// TIA Portal project "Projet_charg_bout" (V15)

(* hardware
DEVICE "PC-System_1"  SIMATIC PC station
   slot 0: "Station PC SIMATIC"  Rail  SIMATIC PC-Station  V1.0
      slot 125: "Stationmanager"  Station_Manager  V6.0.4
   slot 1: "HMI_RT_1"  WinCC RT Advanced  6AV2 104-0xxxx-xxxx  15.0.0.0
      slot 33792: "Interface hôte"  Host interface
   slot 2: "IE Général_1"  IE General  IE_CP  V8.2.0
DEVICE "Station S7-1200_1"  S7-1200 Station
   slot 0: "Châssis_0"  S7-1200 Rack  Rack  V1.0
   slot 1: "PLC_1"  CPU 1214C AC/DC/Rly  6ES7 214-1BG40-0XB0  V4.2
*)

// ===== PLC "PLC_1"  CPU 1214C AC/DC/Rly =====

VAR_GLOBAL   // PLC tag table "Table de variables standard"
   "Tag_1" AT %M100.0 : Bool;
END_VAR

VAR_GLOBAL   // PLC tag table "INPUT"
   "I_GHT" AT %I0.0 : Bool;
   "I_GHD" AT %I0.1 : Bool;
   "I_CB_CHAT" AT %I0.2 : Bool;
   "BI_START" AT %I0.3 : Bool;
   "I_CB_CHAT_TRONG_KET" AT %I0.4 : Bool;
   "M_GHT" AT %M0.0 : Bool;
   "M_GHD" AT %M0.1 : Bool;
   "M_CB_CHAT" AT %M0.2 : Bool;
   "BM_START" AT %M0.3 : Bool;
   "M_CB_CHAT_TRONG_KET" AT %M0.4 : Bool;
   "BM_SIMULATION" AT %M0.5 : Bool;
   "BM_RESET" AT %M0.6 : Bool;
END_VAR

VAR_GLOBAL   // PLC tag table "OUTPUT"
   "Q_VAN_XA" AT %Q0.0 : Bool;
   "Q_HA" AT %Q0.1 : Bool;
   "Q_NAGA" AT %Q0.2 : Bool;
   "Q_BT" AT %Q0.3 : Bool;
   "Q_FULL" AT %Q0.4 : Bool;
END_VAR

VAR_GLOBAL   // PLC tag table "MANU_NHO"
   "DEM_CHAI" AT %MW100 : Int;
   "SIMU_CHAI_CO" AT %MW102 : Int;
   "SIMU_CTAY" AT %MW104 : Int;
   "DEM_CHI_ROT" AT %MW106 : Int;
   "SIMU_CHAI_DA_ROT" AT %MW108 : Int;
END_VAR

VAR_GLOBAL   // PLC tag table "DELAY_TIME"
   "BIT_DELAT_1S" AT %M10.0 : Bool;
   "BIT_DELAY_1S_1" AT %M10.1 : Bool;
   "BIT_DELAY_1S_2" AT %M10.2 : Bool;
   "BIT_DELAY_1S_3" AT %M10.3 : Bool;
   "SIMU_CHAI_SP_CD" AT %M10.4 : Bool;
END_VAR

VAR_GLOBAL   // PLC tag table "LENH_pandn"
   "P1" AT %M20.0 : Bool;
   "P2" AT %M20.1 : Bool;
   "BIT=1" AT %M20.2 : Bool;
   "P3" AT %M20.3 : Bool;
   "P4" AT %M20.4 : Bool;
   "P5" AT %M20.5 : Bool;
   "P6" AT %M20.6 : Bool;
   "P7" AT %M20.7 : Bool;
   "P8" AT %M21.0 : Bool;
   "P9" AT %M21.1 : Bool;
   "P10" AT %M21.2 : Bool;
   "P11" AT %M21.3 : Bool;
   "P12" AT %M21.4 : Bool;
   "N1" AT %M21.5 : Bool;
   "N2" AT %M21.6 : Bool;
   "P13" AT %M21.7 : Bool;
   "P14" AT %M22.0 : Bool;
END_VAR

// folder: System blocks/Program resources

DATA_BLOCK "IEC_Timer_0_DB"   // DB1
{ S7_Optimized_Access := 'TRUE' }
AUTHOR : Simatic
FAMILY : IEC
NAME : IEC_TMR
VERSION : 1.0
// stored: InstanceOfName IEC_TIMER
"IEC_TIMER"
BEGIN
END_DATA_BLOCK

DATA_BLOCK "IEC_Timer_0_DB_1"   // DB2
{ S7_Optimized_Access := 'TRUE' }
AUTHOR : Simatic
FAMILY : IEC
NAME : IEC_TMR
VERSION : 1.0
// stored: InstanceOfName IEC_TIMER
"IEC_TIMER"
BEGIN
END_DATA_BLOCK

DATA_BLOCK "IEC_Timer_0_DB_2"   // DB3
{ S7_Optimized_Access := 'TRUE' }
AUTHOR : Simatic
FAMILY : IEC
NAME : IEC_TMR
VERSION : 1.0
// stored: InstanceOfName IEC_TIMER
"IEC_TIMER"
BEGIN
END_DATA_BLOCK

DATA_BLOCK "IEC_Timer_0_DB_3"   // DB4
{ S7_Optimized_Access := 'TRUE' }
AUTHOR : Simatic
FAMILY : IEC
NAME : IEC_TMR
VERSION : 1.0
// stored: InstanceOfName IEC_TIMER
"IEC_TIMER"
BEGIN
END_DATA_BLOCK

DATA_BLOCK "IEC_Timer_0_DB_4"   // DB5
{ S7_Optimized_Access := 'TRUE' }
AUTHOR : Simatic
FAMILY : IEC
NAME : IEC_TMR
VERSION : 1.0
// stored: InstanceOfName IEC_TIMER
"IEC_TIMER"
BEGIN
END_DATA_BLOCK

DATA_BLOCK "IEC_Timer_0_DB_5"   // DB6
{ S7_Optimized_Access := 'TRUE' }
AUTHOR : Simatic
FAMILY : IEC
NAME : IEC_TMR
VERSION : 1.0
// stored: InstanceOfName IEC_TIMER
"IEC_TIMER"
BEGIN
END_DATA_BLOCK

DATA_BLOCK "IEC_Timer_0_DB_6"   // DB7
{ S7_Optimized_Access := 'TRUE' }
AUTHOR : Simatic
FAMILY : IEC
NAME : IEC_TMR
VERSION : 1.0
// stored: InstanceOfName IEC_TIMER
"IEC_TIMER"
BEGIN
END_DATA_BLOCK

// folder: (top level)

FUNCTION "FC_SUMILATION" : Void   // FC1, LAD
{ S7_Optimized_Access := 'TRUE' }
VERSION : 0.1
   VAR_TEMP   // added for the SCL form of the ladder/FBD networks
      _w1 : Bool;
   END_VAR
BEGIN

REGION Network 1
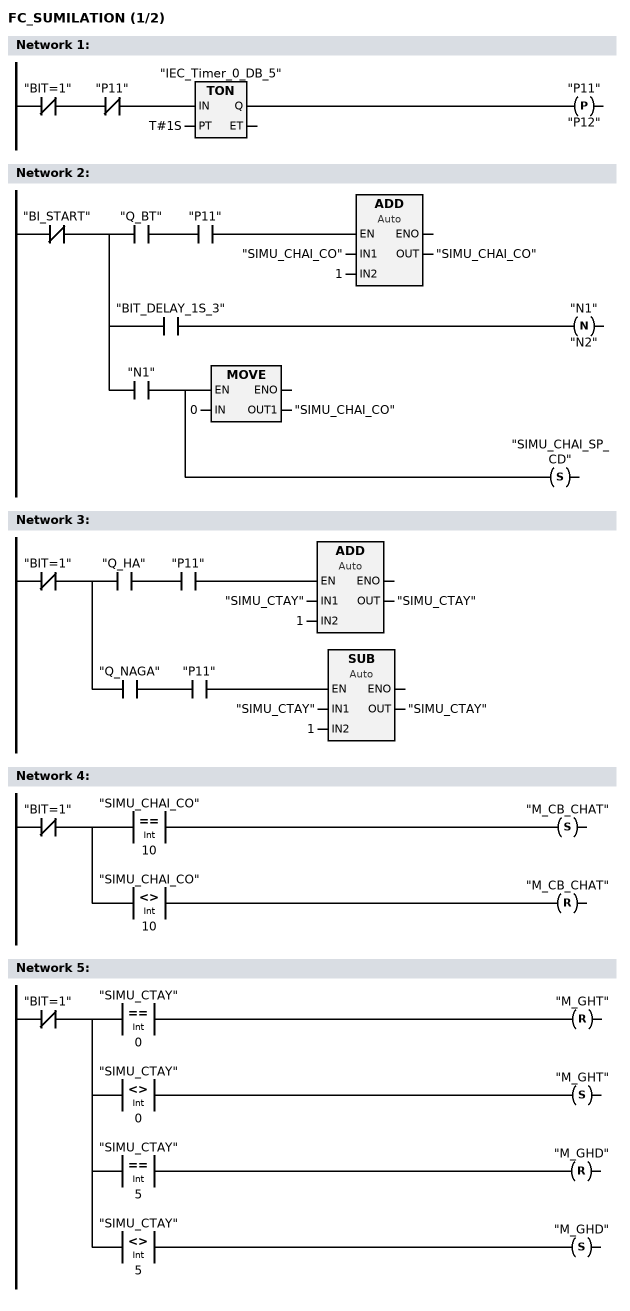
   "IEC_Timer_0_DB_5".TON(IN := NOT "BIT=1" AND NOT "P11", PT := T#1S);
   "P11" := "IEC_Timer_0_DB_5".Q AND NOT "P12";   // rising edge
   "P12" := "IEC_Timer_0_DB_5".Q;
END_REGION

REGION Network 2
   IF NOT "BI_START" AND "Q_BT" AND "P11" THEN "SIMU_CHAI_CO" := "SIMU_CHAI_CO" + 1; END_IF;
   #_w1 := NOT "BI_START" AND "BIT_DELAY_1S_3";
   "N1" := NOT #_w1 AND "N2";   // falling edge
   "N2" := #_w1;
   IF NOT "BI_START" AND "N1" THEN
       "SIMU_CHAI_CO" := 0;
       "SIMU_CHAI_SP_CD" := TRUE;
   END_IF;
END_REGION

REGION Network 3
   RUNG wire#powerrail
      I_Contact( "BIT=1" )
      wire#w1
      Contact( "Q_HA" )
      Contact( "P11" )
      Add(in1 := "SIMU_CTAY", in2 := 1, out => "SIMU_CTAY")
   END_RUNG
   RUNG wire#w1
      Contact( "Q_NAGA" )
      Contact( "P11" )
      Sub(in1 := "SIMU_CTAY", in2 := 1, out => "SIMU_CTAY")
   END_RUNG
   // the same network as SCL:
   IF NOT "BIT=1" AND "Q_HA" AND "P11" THEN "SIMU_CTAY" := "SIMU_CTAY" + 1; END_IF;
   IF NOT "BIT=1" AND "Q_NAGA" AND "P11" THEN "SIMU_CTAY" := "SIMU_CTAY" - 1; END_IF;
END_REGION

REGION Network 4
   RUNG wire#powerrail
      I_Contact( "BIT=1" )
      wire#w1
      { S7_Templates := "SrcType := Int" } EQ_Contact(in1 := "SIMU_CHAI_CO", in2 := 10)
      S_Coil( "M_CB_CHAT" )
   END_RUNG
   RUNG wire#w1
      { S7_Templates := "SrcType := Int" } NE_Contact(in1 := "SIMU_CHAI_CO", in2 := 10)
      R_Coil( "M_CB_CHAT" )
   END_RUNG
   // the same network as SCL:
   IF NOT "BIT=1" AND ("SIMU_CHAI_CO" = 10) THEN "M_CB_CHAT" := TRUE; END_IF;
   IF NOT "BIT=1" AND ("SIMU_CHAI_CO" <> 10) THEN "M_CB_CHAT" := FALSE; END_IF;
END_REGION

REGION Network 5
   RUNG wire#powerrail
      I_Contact( "BIT=1" )
      wire#w1
      { S7_Templates := "SrcType := Int" } EQ_Contact(in1 := "SIMU_CTAY", in2 := 0)
      R_Coil( "M_GHT" )
   END_RUNG
   RUNG wire#w1
      { S7_Templates := "SrcType := Int" } NE_Contact(in1 := "SIMU_CTAY", in2 := 0)
      S_Coil( "M_GHT" )
   END_RUNG
   RUNG wire#w1
      { S7_Templates := "SrcType := Int" } EQ_Contact(in1 := "SIMU_CTAY", in2 := 5)
      R_Coil( "M_GHD" )
   END_RUNG
   RUNG wire#w1
      { S7_Templates := "SrcType := Int" } NE_Contact(in1 := "SIMU_CTAY", in2 := 5)
      S_Coil( "M_GHD" )
   END_RUNG
   // the same network as SCL:
   IF NOT "BIT=1" AND ("SIMU_CTAY" = 0) THEN "M_GHT" := FALSE; END_IF;
   IF NOT "BIT=1" AND ("SIMU_CTAY" <> 0) THEN "M_GHT" := TRUE; END_IF;
   IF NOT "BIT=1" AND ("SIMU_CTAY" = 5) THEN "M_GHD" := FALSE; END_IF;
   IF NOT "BIT=1" AND ("SIMU_CTAY" <> 5) THEN "M_GHD" := TRUE; END_IF;
END_REGION

REGION Network 6
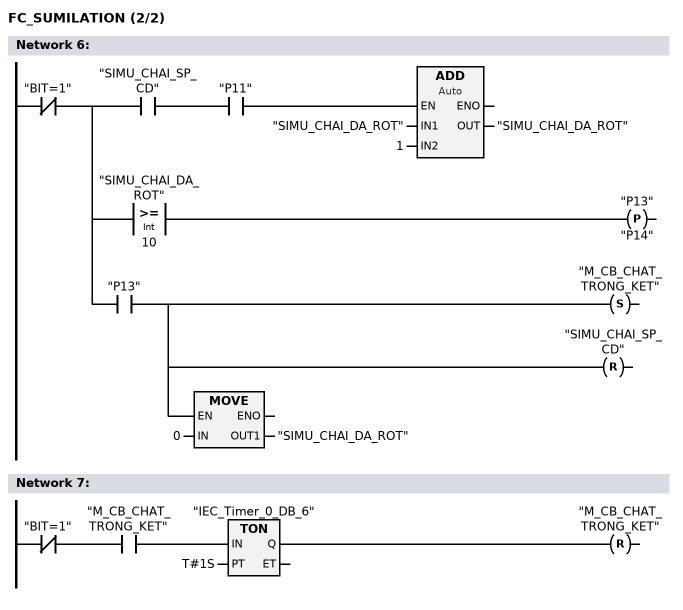
   IF NOT "BIT=1" AND "SIMU_CHAI_SP_CD" AND "P11" THEN "SIMU_CHAI_DA_ROT" := "SIMU_CHAI_DA_ROT" + 1; END_IF;
   #_w1 := NOT "BIT=1" AND ("SIMU_CHAI_DA_ROT" >= 10);
   "P13" := #_w1 AND NOT "P14";   // rising edge
   "P14" := #_w1;
   IF NOT "BIT=1" AND "P13" THEN
       "M_CB_CHAT_TRONG_KET" := TRUE;
       "SIMU_CHAI_SP_CD" := FALSE;
       "SIMU_CHAI_DA_ROT" := 0;
   END_IF;
END_REGION

REGION Network 7
   "IEC_Timer_0_DB_6".TON(IN := NOT "BIT=1" AND "M_CB_CHAT_TRONG_KET", PT := T#1S);
   IF "IEC_Timer_0_DB_6".Q THEN "M_CB_CHAT_TRONG_KET" := FALSE; END_IF;
END_REGION
END_FUNCTION

ORGANIZATION_BLOCK "Main"   // OB1, LAD, ProgramCycle
TITLE = "Main Program Sweep (Cycle)"
{ S7_Optimized_Access := 'TRUE' }
VERSION : 0.1
   VAR_INPUT
      Initial_Call : Bool;   // Initial call of this OB
      Remanence : Bool;   // =True, if remanent data are available
   END_VAR
   VAR_TEMP   // added for the SCL form of the ladder/FBD networks
      _w1 : Bool;
      _w2 : Bool;
   END_VAR
BEGIN

REGION Network 1
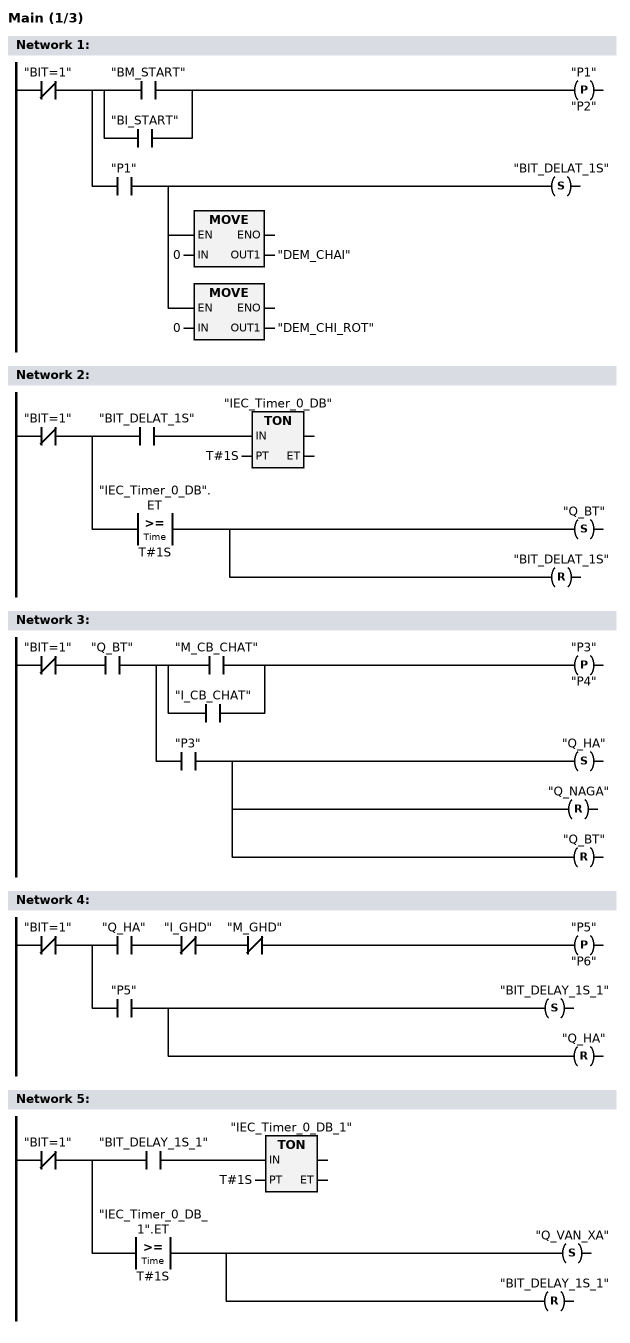
   #_w1 := NOT "BIT=1" AND ("BM_START" OR "BI_START");
   "P1" := #_w1 AND NOT "P2";   // rising edge
   "P2" := #_w1;
   IF NOT "BIT=1" AND "P1" THEN
       "BIT_DELAT_1S" := TRUE;
       "DEM_CHAI" := 0;
       "DEM_CHI_ROT" := 0;
   END_IF;
END_REGION

REGION Network 2
   "IEC_Timer_0_DB".TON(IN := NOT "BIT=1" AND "BIT_DELAT_1S", PT := T#1S);
   IF NOT "BIT=1" AND ("IEC_Timer_0_DB".ET >= T#1S) THEN
       "Q_BT" := TRUE;
       "BIT_DELAT_1S" := FALSE;
   END_IF;
END_REGION

REGION Network 3
   #_w1 := NOT "BIT=1" AND "Q_BT";
   #_w2 := #_w1 AND ("M_CB_CHAT" OR "I_CB_CHAT");
   "P3" := #_w2 AND NOT "P4";   // rising edge
   "P4" := #_w2;
   IF #_w1 AND "P3" THEN
       "Q_HA" := TRUE;
       "Q_NAGA" := FALSE;
       "Q_BT" := FALSE;
   END_IF;
END_REGION

REGION Network 4
   #_w1 := NOT "BIT=1" AND "Q_HA" AND NOT "I_GHD" AND NOT "M_GHD";
   "P5" := #_w1 AND NOT "P6";   // rising edge
   "P6" := #_w1;
   IF NOT "BIT=1" AND "P5" THEN
       "BIT_DELAY_1S_1" := TRUE;
       "Q_HA" := FALSE;
   END_IF;
END_REGION

REGION Network 5
   "IEC_Timer_0_DB_1".TON(IN := NOT "BIT=1" AND "BIT_DELAY_1S_1", PT := T#1S);
   IF NOT "BIT=1" AND ("IEC_Timer_0_DB_1".ET >= T#1S) THEN
       "Q_VAN_XA" := TRUE;
       "BIT_DELAY_1S_1" := FALSE;
   END_IF;
END_REGION

REGION Network 6
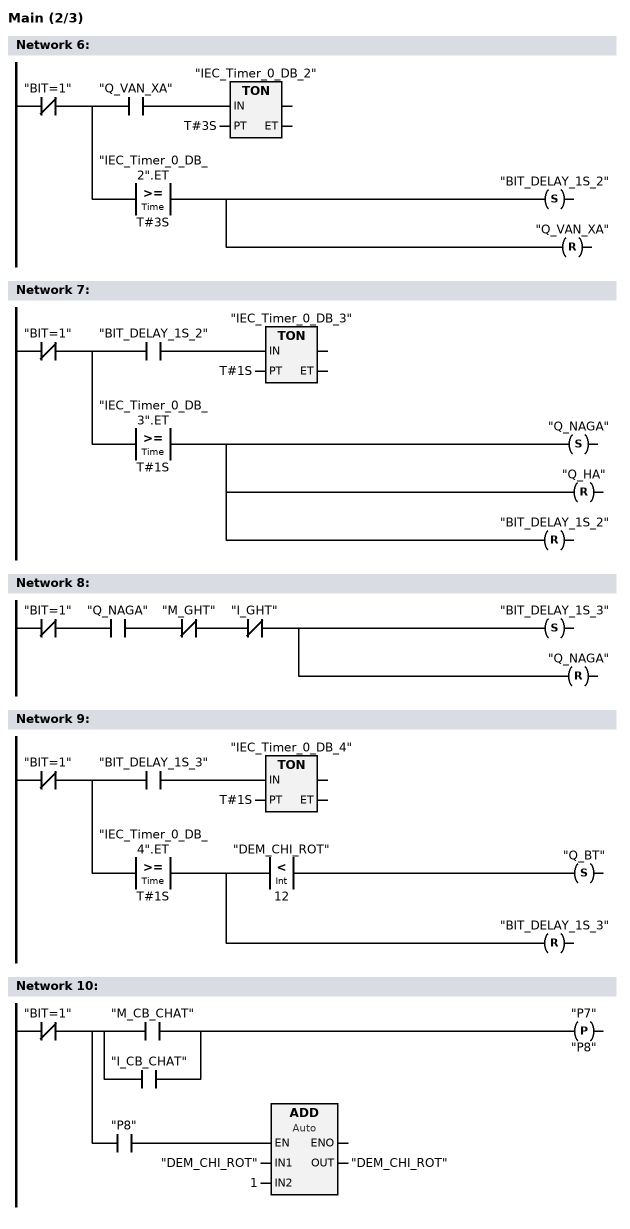
   "IEC_Timer_0_DB_2".TON(IN := NOT "BIT=1" AND "Q_VAN_XA", PT := T#3S);
   IF NOT "BIT=1" AND ("IEC_Timer_0_DB_2".ET >= T#3S) THEN
       "BIT_DELAY_1S_2" := TRUE;
       "Q_VAN_XA" := FALSE;
   END_IF;
END_REGION

REGION Network 7
   "IEC_Timer_0_DB_3".TON(IN := NOT "BIT=1" AND "BIT_DELAY_1S_2", PT := T#1S);
   IF NOT "BIT=1" AND ("IEC_Timer_0_DB_3".ET >= T#1S) THEN
       "Q_NAGA" := TRUE;
       "Q_HA" := FALSE;
       "BIT_DELAY_1S_2" := FALSE;
   END_IF;
END_REGION

REGION Network 8
   RUNG wire#powerrail
      I_Contact( "BIT=1" )
      Contact( "Q_NAGA" )
      I_Contact( "M_GHT" )
      I_Contact( "I_GHT" )
      wire#w1
      S_Coil( "BIT_DELAY_1S_3" )
   END_RUNG
   RUNG wire#w1
      R_Coil( "Q_NAGA" )
   END_RUNG
   // the same network as SCL:
   IF NOT "BIT=1" AND "Q_NAGA" AND NOT "M_GHT" AND NOT "I_GHT" THEN
       "BIT_DELAY_1S_3" := TRUE;
       "Q_NAGA" := FALSE;
   END_IF;
END_REGION

REGION Network 9
   "IEC_Timer_0_DB_4".TON(IN := NOT "BIT=1" AND "BIT_DELAY_1S_3", PT := T#1S);
   #_w1 := NOT "BIT=1" AND ("IEC_Timer_0_DB_4".ET >= T#1S);
   IF #_w1 AND ("DEM_CHI_ROT" < 12) THEN "Q_BT" := TRUE; END_IF;
   IF #_w1 THEN "BIT_DELAY_1S_3" := FALSE; END_IF;
END_REGION

REGION Network 10
   #_w1 := NOT "BIT=1" AND ("M_CB_CHAT" OR "I_CB_CHAT");
   "P7" := #_w1 AND NOT "P8";   // rising edge
   "P8" := #_w1;
   IF NOT "BIT=1" AND "P8" THEN "DEM_CHI_ROT" := "DEM_CHI_ROT" + 1; END_IF;
END_REGION

REGION Network 11
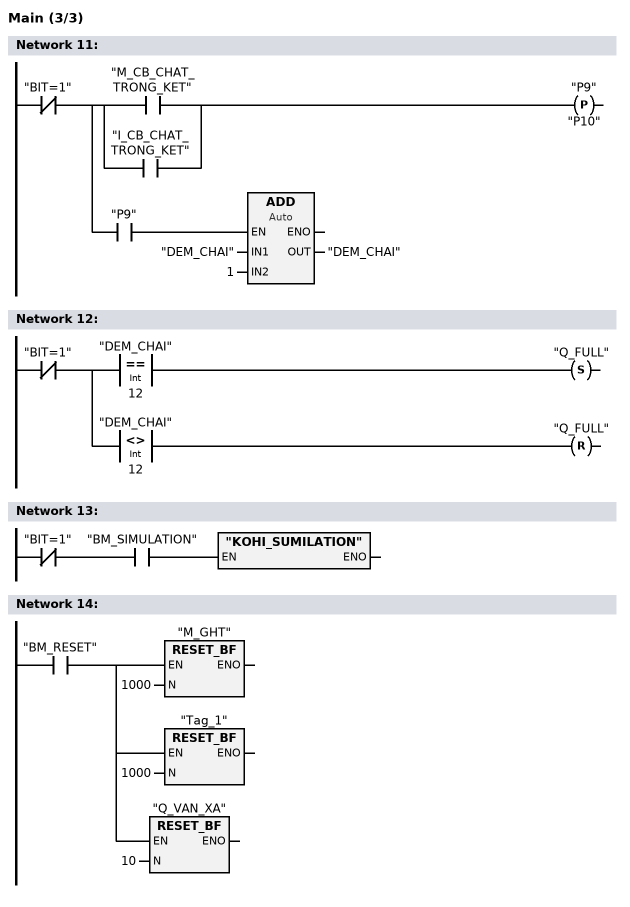
   #_w1 := NOT "BIT=1" AND ("M_CB_CHAT_TRONG_KET" OR "I_CB_CHAT_TRONG_KET");
   "P9" := #_w1 AND NOT "P10";   // rising edge
   "P10" := #_w1;
   IF NOT "BIT=1" AND "P9" THEN "DEM_CHAI" := "DEM_CHAI" + 1; END_IF;
END_REGION

REGION Network 12
   RUNG wire#powerrail
      I_Contact( "BIT=1" )
      wire#w1
      { S7_Templates := "SrcType := Int" } EQ_Contact(in1 := "DEM_CHAI", in2 := 12)
      S_Coil( "Q_FULL" )
   END_RUNG
   RUNG wire#w1
      { S7_Templates := "SrcType := Int" } NE_Contact(in1 := "DEM_CHAI", in2 := 12)
      R_Coil( "Q_FULL" )
   END_RUNG
   // the same network as SCL:
   IF NOT "BIT=1" AND ("DEM_CHAI" = 12) THEN "Q_FULL" := TRUE; END_IF;
   IF NOT "BIT=1" AND ("DEM_CHAI" <> 12) THEN "Q_FULL" := FALSE; END_IF;
END_REGION

REGION Network 13
   RUNG wire#powerrail
      I_Contact( "BIT=1" )
      Contact( "BM_SIMULATION" )
      "KOHI_SUMILATION"()
   END_RUNG
   // the same network as SCL:
   IF NOT "BIT=1" AND "BM_SIMULATION" THEN "KOHI_SUMILATION"(); END_IF;
END_REGION

REGION Network 14
   // no SCL statement known for RBitfield: written as a call
   #_w1 := "BM_RESET";
   IF #_w1 THEN
       RESET_BF(operand := "M_GHT", n := 1000);
       RESET_BF(operand := "Tag_1", n := 1000);
       RESET_BF(operand := "Q_VAN_XA", n := 10);
   END_IF;
END_REGION
END_ORGANIZATION_BLOCK

(* ===== HMI "HMI_RT_1" =====
system functions are stored by id; their names below are inferred from use
connection "HMI_Liaison_1": ETHERNET, S7_1200_OMS

HMI tags "Table de variables standard"
   "DEM_CHAI" : Int = PLC DEM_CHAI AT %MW100, 1 s
   "Q_VAN_XA" : Bool = PLC Q_VAN_XA AT %Q0.0, 1 s
   "M_GHT" : Bool = PLC M_GHT AT %M0.0, 1 s
   "M_GHD" : Bool = PLC M_GHD AT %M0.1, 1 s
   "M_CB_CHAT" : Bool = PLC M_CB_CHAT AT %M0.2, 1 s
   "M_CB_CHAT_TRONG_KET" : Bool = PLC M_CB_CHAT_TRONG_KET AT %M0.4, 1 s
   "Q_BT" : Bool = PLC Q_BT AT %Q0.3, 1 s
   "Q_HA" : Bool = PLC Q_HA AT %Q0.1, 1 s
   "Q_NAGA" : Bool = PLC Q_NAGA AT %Q0.2, 1 s
   "Q_FULL" : Bool = PLC Q_FULL AT %Q0.4, 1 s
   "DEM_CHI_ROT" : Int = PLC DEM_CHI_ROT AT %MW106, 1 s
   "SIMU_CHAI_CO" : Int = PLC SIMU_CHAI_CO AT %MW102, 1 s
   "SIMU_CHAI_DA_ROT" : Int = PLC SIMU_CHAI_DA_ROT AT %MW108, 1 s
   "SIMU_CTAY" : Int = PLC SIMU_CTAY AT %MW104, 1 s
   "BM_START" : Bool = PLC BM_START AT %M0.3, 1 s
   "BM_SIMULATION" : Bool = PLC BM_SIMULATION AT %M0.5, 1 s
   "BM_RESET" : Bool = PLC BM_RESET AT %M0.6, 1 s
   "SIMU_CHAI_SP_CD" : Bool = PLC SIMU_CHAI_SP_CD AT %M10.4, 1 s

screen "Vue_1" 800x1280
   SymbolLibrary "Bibliothèque des icônes_18" at 326,31 size 13x211
   SymbolLibrary "Bibliothèque des icônes_19" at 311,119 size 28x31
   SymbolLibrary "Bibliothèque des icônes_20" at 240,128 size 75x13
   SymbolLibrary "Bibliothèque des icônes_21" at 311,189 size 28x31
   SymbolLibrary "Bibliothèque des icônes_22" at 239,198 size 75x13
   SymbolLibrary "Bibliothèque des icônes_23" at 321,56 size 54x44
      Appearance <- "Q_VAN_XA"
   SymbolLibrary "Bibliothèque des icônes_26" at 233,95 size 30x142
   Rectangle "Rectangle_2" at 502,52 size 21x49
      Appearance <- "Q_HA"
      Visibility <- "Q_HA"
   Polygon "Polygone_1" at 492,94 size 42x25
      Appearance <- "Q_HA"
      Visibility <- "Q_HA"
   Rectangle "Rectangle_3" at 502,84 size 21x49
      Visibility <- "Q_NAGA"
      Appearance <- "Q_NAGA"
   Polygon "Polygone_2" at 492,52 size 42x32
      Visibility <- "Q_NAGA"
      Appearance <- "Q_NAGA"
   SymbolLibrary "Bibliothèque des icônes_1" at 14,287 size 323x51
      Appearance <- "Q_BT"
   SymbolLibrary "Bibliothèque des icônes_9" at 280,287 size 323x51
      Appearance <- "Q_BT"
   SymbolLibrary "Bibliothèque des icônes_10" at 349,104 size 58x24
      Appearance <- "M_GHT"
   SymbolLibrary "Bibliothèque des icônes_11" at 350,168 size 58x24
      Appearance <- "M_GHD"
   SymbolLibrary "Bibliothèque des icônes_12" at 322,318 size 27x54
      Appearance <- "M_CB_CHAT"
   SymbolLibrary "Bibliothèque des icônes_13" at 63,247 size 27x54
      HorizontalMovement <- "SIMU_CHAI_CO"
   SymbolLibrary "Bibliothèque des icônes_14" at 552,321 size 124x54
   Circle "Cercle_1" at 553,84 size 30x30
      Visibility <- "DEM_CHAI"
   Circle "Cercle_2" at 604,85 size 30x30
      Visibility <- "DEM_CHAI"
   Circle "Cercle_3" at 657,84 size 30x30
      Visibility <- "DEM_CHAI"
   Circle "Cercle_4" at 553,114 size 30x30
      Visibility <- "DEM_CHAI"
   Circle "Cercle_5" at 604,115 size 30x30
      Visibility <- "DEM_CHAI"
   Circle "Cercle_6" at 657,114 size 30x30
      Visibility <- "DEM_CHAI"
   Circle "Cercle_7" at 553,144 size 30x30
      Visibility <- "DEM_CHAI"
   Circle "Cercle_8" at 604,145 size 30x30
      Visibility <- "DEM_CHAI"
   Circle "Cercle_9" at 657,144 size 30x30
      Visibility <- "DEM_CHAI"
   Circle "Cercle_10" at 553,174 size 30x30
      Visibility <- "DEM_CHAI"
   Circle "Cercle_11" at 604,175 size 30x30
      Visibility <- "DEM_CHAI"
   Circle "Cercle_12" at 657,174 size 30x30
      Visibility <- "DEM_CHAI"
   TextField "Champ de texte_1" at 424,104 size 36x22; Text 'GHT'
   TextField "Champ de texte_2" at 424,171 size 38x22; Text 'GHD'
   SymbolLibrary "Bibliothèque des icônes_15" at 666,338 size 27x54
      Appearance <- "M_CB_CHAT_TRONG_KET"
   SymbolLibrary "Bibliothèque des icônes_17" at 319,247 size 26x53
      HorizontalMovement <- "SIMU_CHAI_DA_ROT"
      Visibility <- "SIMU_CHAI_SP_CD"
   SymbolLibrary "Bibliothèque des icônes_16" at 44,358 size 73x63
      Appearance <- "Q_BT"
   Group "Group" at 239,31 size 136x211
      VerticalMovement <- "SIMU_CTAY"
   Group "Group_2" at 492,52 size 42x81
   Circle "Cercle_13" at 879,239 size 40x40
      Appearance <- "Q_FULL"
   IOField "Champ d'E/S_1" at 296,382 size 63x35; FormatPattern s999
      ProcessValue <- "DEM_CHI_ROT"
   IOField "Champ d'E/S_2" at 643,411 size 63x35; FormatPattern s999
      ProcessValue <- "DEM_CHAI"
   IOField "Champ d'E/S_3" at 585,205 size 63x35; FormatPattern s999
      ProcessValue <- "DEM_CHAI"
   Button "Bouton_1" at 49,91 size 88x37; TextOff 'START'
      on Press: SetBit("BM_START")
      on Release: ResetBit("BM_START")
   Button "Bouton_2" at 49,132 size 88x37; TextOff 'SIMU ON'
      on Press: SetBit("BM_SIMULATION")
      Appearance <- "BM_SIMULATION"
   Button "Bouton_3" at 48,175 size 88x37; TextOff 'SIMU OFF'
      on Press: ResetBit("BM_SIMULATION")
   Button "Bouton_4" at 49,52 size 88x37; TextOff 'RESET'
      on Press: SetBit("BM_RESET")
   Group "Group_1" at 492,52 size 42x67
*)